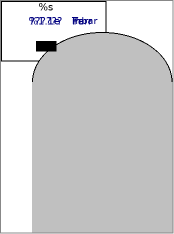
VISUALIZATION VISU_JAUGE_PCG550_ETHERCAT  // 174x234
VAR_IN_OUT
	m_Input_JAUGE:		BLOCK_PCG550_ETHERCAT;
END_VAR
    Rectangle (1,1 105x60), invisible if: TRUE
    Rectangle (1,11 90x20), "??????", invisible if: (m_Input_JAUGE.STATE_OK) <> 0
    Group (32,32 28x28)
        Ellipse (0,0 140x100)
        Rectangle (0,50 140x150)
        Polyline (140,50)
    Rectangle (36,41 20x10), colour toggle: TRUE
    Rectangle (11,2 70x10), "%s", text variable: m_Input_JAUGE.MNEMO
    Group (6,11 88x18), invisible if: NOT m_Input_JAUGE.STATE_OK
        Rectangle (0,0 57x20), "%1.1e", text variable: m_Input_JAUGE.STATE_Pression
        Rectangle (60,0 27x20), "Torr", invisible if: NOT (m_Input_JAUGE.CONF_unit = 1)
        Rectangle (60,0 30x20), "mbar", invisible if: NOT (m_Input_JAUGE.CONF_unit = 0)
        Rectangle (60,0 27x20), "Pa", invisible if: NOT (m_Input_JAUGE.CONF_unit = 2)
END_VISUALIZATION

(* stored: Version 1.1.0.1, ProductVersion 3.1.4024.10
   Visu VISU_JAUGE_PCG550_ETHERCAT: Id {322f5cac-ad61-4c0f-bd0f-939aa94ae1d5} *)
